FUNCTION_BLOCK ProductBase EXTENDS HardwareObservationBase
VAR CONSTANT
	RES_IDX: UINT := 0;
END_VAR
VAR
	// ***** MODIFIED BY RA *****
	raIn_isRemote: BOOL;
	raIn_prodTypeAdr: SAdsSymbol;	// points to the remote's product type (at m_vals[RES_IDX].Values.Numeric)
	raIn_copiedTypeAdr: SAdsSymbol;	// points to the remote's m_copiedProdType
	raIn_resetAdr: SAdsSymbol;		// points to the remote's reset flag
	// **************************
	
	// ***** INIT BY RA OR SUBCLASS *****
	raIn_processStateIdx: UINT;
	// **********************************

	// an array of values characterizing the product. At RES_IDX=0, there is an aggregated "product type"
	m_vals: ARRAY [ResiConst.ARR_MIN..ResiConst.DEFAULT_ARR_MAX] OF SValue;
	// a number (may be an ENUM) defining the type of product. NOTE: 0 means null/nil/None.
	m_copiedProdType: LREAL;
	
	m_valReader: ADSREAD;
	m_copyTrigWriter: ADSWRITE;
	m_resetWriter: ADSWRITE;
	
	// flags
	m_resetPending: BOOL;
	m_defResetPending: BOOL;
	m_trueVal: BOOL := TRUE;
END_VAR

METHOD Copy : BOOL
VAR_INPUT
	i_ptrOther: POINTER TO ProductBase;
END_VAR
Copy := FALSE;

IF NOT raIn_isRemote THEN
	m_copiedProdType := i_ptrOther^.m_vals[RES_IDX].Value.Numeric;
ELSE
	// trigger the remote to do a copy operation
	m_copyTrigWriter(
		NETID := raIn_copiedTypeAdr.NetId,
		PORT := raIn_copiedTypeAdr.Port,
		IDXGRP := raIn_copiedTypeAdr.IdxGrp,
		IDXOFFS := raIn_copiedTypeAdr.IdxOffs,
		LEN := SIZEOF(i_ptrOther^.m_vals[RES_IDX].Value.Numeric),
		SRCADDR := ADR(i_ptrOther^.m_vals[RES_IDX].Value.Numeric),
		WRITE := TRUE);
END_IF

IF NOT m_copyTrigWriter.BUSY THEN
	m_copyTrigWriter(WRITE := FALSE);
	Copy := TRUE;
END_IF
END_METHOD

METHOD Reset : BOOL
m_resetPending := TRUE;
END_METHOD

METHOD ResetConfiguration : BOOL
VAR
	emptySym: SAdsSymbol;
END_VAR
raIn_processStateIdx := 0;

raIn_copiedTypeAdr := emptySym;
raIn_prodTypeAdr := emptySym;
raIn_resetAdr := emptySym;
END_METHOD

METHOD ResetDefinition : BOOL
m_defResetPending := TRUE;
END_METHOD

(* Based on the aggregated product type value, set the separete input values for a consistent shift register. *)
METHOD ReverseSetInputs : BOOL
// not required for the ProductBase
END_METHOD

(* Update an instance of ProcessState with the part of the process that can be observed by this Hardware Interface. *)
METHOD UpdateProcessObservation : BOOL
VAR_IN_OUT
	io_processState: ProcessState;
END_VAR
VAR
	emptyVals: ARRAY [ResiConst.ARR_MIN..ResiConst.DEFAULT_ARR_MAX] OF SValue;
END_VAR
IF raIn_processStateIdx = 0 OR m_copyTrigWriter.BUSY THEN
	RETURN;
END_IF

IF m_copiedProdType <> 0 THEN
	m_vals[RES_IDX].Defined := TRUE;
	m_vals[RES_IDX].DataType := EDataType.numeric;
	m_vals[RES_IDX].Value.Numeric := m_copiedProdType;
	
	ReverseSetInputs();
	m_copiedProdType := 0;
END_IF

// synchronize with the StateTracker's state
UpdateProcessObsInternal(io_processState);

// deal with reset requests
m_resetWriter();	// read takes multiple cycles
IF m_resetPending THEN
	IF raIn_isRemote THEN
		// set the remote's reset flag (the local instance will be synced below)
		m_resetWriter(WRITE := FALSE);
		m_resetWriter(
			NETID := raIn_resetAdr.NetId,
			PORT := raIn_resetAdr.Port,
			IDXGRP := raIn_resetAdr.IdxGrp,
			IDXOFFS := raIn_resetAdr.IdxOffs,
			LEN := SIZEOF(m_trueVal),
			SRCADDR := ADR(m_trueVal),
			WRITE := TRUE);
	ELSE
		m_vals[RES_IDX].Value.Numeric := 0;
		ReverseSetInputs();
	END_IF
	
	m_resetPending := FALSE;
	RETURN;
END_IF

// update this product base with the remote's value
IF raIn_isRemote THEN
	// TODO - other data types and potentially multiple result values
	m_vals[RES_IDX].Defined := TRUE;
	m_vals[RES_IDX].DataType := EDataType.numeric;

	m_valReader(READ := FALSE);
	m_valReader(
		NETID := raIn_prodTypeAdr.NetId,
		PORT := raIn_prodTypeAdr.Port,
		IDXGRP := raIn_prodTypeAdr.IdxGrp,
		IDXOFFS := raIn_prodTypeAdr.IdxOffs,
		LEN := SIZEOF(m_vals[RES_IDX].Value.Numeric),
		DESTADDR := ADR(m_vals[RES_IDX].Value.Numeric),
		READ := TRUE);
END_IF
END_METHOD

METHOD PROTECTED UpdateProcessObsInternal : BOOL
VAR_IN_OUT
	io_processState: ProcessState;
END_VAR
// not required for the ProductBase
END_METHOD

END_FUNCTION_BLOCK

(* stored: Version 1.1.0.1
   POU ProductBase: Id {0215d773-ad29-488c-b3e2-f619c5307d05}, SpecialFunc None
   Method Copy: Id {f6d699f0-d197-47e5-8b2c-dc7ccca00b23}
   Method Reset: Id {8e74e174-b0a7-4f71-8dbb-0aae7e39d580}
   Method ResetConfiguration: Id {94f2bc4d-8302-4541-ad8c-fc961d758187}
   Method ResetDefinition: Id {71a74ce8-9db8-447e-9533-403e2cbc5224}
   Method ReverseSetInputs: Id {1b852751-0370-4a10-b861-bfbff8021f35}
   Method UpdateProcessObservation: Id {39e5fe45-bc3d-41f1-a7c7-9f9faad16085}
   Method UpdateProcessObsInternal: Id {4a63e994-68a0-432c-a803-4f1f9a1f4f29} *)
